TYPE U_ReinterpretDALIEnum :
UNION
	raw				: BYTE;
	eventScheme 	: E_DALIEventScheme;
	fadeTime		: E_DALIFadeTime;
	testTiming      : E_DALITestTiming;
END_UNION
END_TYPE

(* stored: Version 1.1.0.1, ProductVersion 3.1.4024.11
   DUT U_ReinterpretDALIEnum: Id {4b3b4271-a73b-4033-bd66-391eb231e809} *)
